// TIA Portal project "Elevator" (V16)

(* hardware
DEVICE "S71500/ET200MP station_1"  S7-1500 station
   slot 0: "Perfil soporte_0"  Rack  6ES7 590-1***0-0AA0
   slot 1: "PLC_1"  CPU 1511-1 PN  6ES7 511-1AK02-0AB0  V2.8
      slot 3: "Display de la CPU_1"  6ES7591-1AA00-0AA0
      slot 32768: "Interfaz PROFINET_1"  X1
         slot 32769: "Puerto_1"  X1 P1
         slot 32770: "Puerto_2"  X1 P2
      slot 34817: "Virtual CP interface port_1"  Virtual CP interface port  Virtual CP interface port
*)

// ===== PLC "PLC_1"  CPU 1511-1 PN =====

VAR_GLOBAL   // PLC tag table "Tabla de variables estándar"
   "Tag_1" AT %M0.0 : Bool;
   "Tag_2" AT %M0.1 : Bool;
   "Tag_3" AT %M200.0 : Bool;
END_VAR

DATA_BLOCK "Floor"   // DB1
{ S7_Optimized_Access := 'TRUE' }
VERSION : 0.1
   VAR
      Piso_1 : Real := 3166.0;
      Piso_2 : Real := 6332.0;
      Piso_3 : Real := 9498.0;
      Piso_4 : Real := 12664.0;
      Piso_5 : Real;
      Piso_6 : Real := -19000.0;
      PisoActual : Real := 3166.0;
      Floor_Command : Int := 0;
   END_VAR
BEGIN
END_DATA_BLOCK

ORGANIZATION_BLOCK "Main"   // OB1, LAD, ProgramCycle
TITLE = "Main Program Sweep (Cycle)"
{ S7_Optimized_Access := 'TRUE' }
VERSION : 0.1
   VAR_INPUT
      Initial_Call : Bool;   // Initial call of this OB
      Remanence : Bool;   // =True, if remanent data are available
   END_VAR
BEGIN

REGION Network 1
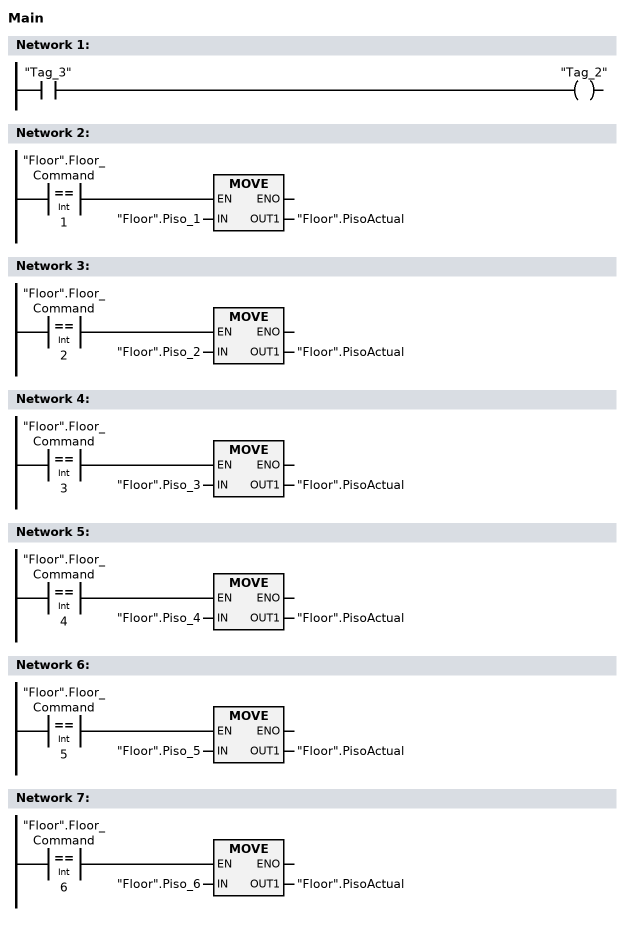
   RUNG wire#powerrail
      Contact( "Tag_3" )
      Coil( "Tag_2" )
   END_RUNG
   // the same network as SCL:
   "Tag_2" := "Tag_3";
END_REGION

REGION Network 2
   RUNG wire#powerrail
      { S7_Templates := "SrcType := Int" } EQ_Contact(in1 := "Floor".Floor_Command, in2 := 1)
      Move(in := "Floor".Piso_1, out1 => "Floor".PisoActual)
   END_RUNG
   // the same network as SCL:
   IF "Floor".Floor_Command = 1 THEN "Floor".PisoActual := "Floor".Piso_1; END_IF;
END_REGION

REGION Network 3
   RUNG wire#powerrail
      { S7_Templates := "SrcType := Int" } EQ_Contact(in1 := "Floor".Floor_Command, in2 := 2)
      Move(in := "Floor".Piso_2, out1 => "Floor".PisoActual)
   END_RUNG
   // the same network as SCL:
   IF "Floor".Floor_Command = 2 THEN "Floor".PisoActual := "Floor".Piso_2; END_IF;
END_REGION

REGION Network 4
   RUNG wire#powerrail
      { S7_Templates := "SrcType := Int" } EQ_Contact(in1 := "Floor".Floor_Command, in2 := 3)
      Move(in := "Floor".Piso_3, out1 => "Floor".PisoActual)
   END_RUNG
   // the same network as SCL:
   IF "Floor".Floor_Command = 3 THEN "Floor".PisoActual := "Floor".Piso_3; END_IF;
END_REGION

REGION Network 5
   RUNG wire#powerrail
      { S7_Templates := "SrcType := Int" } EQ_Contact(in1 := "Floor".Floor_Command, in2 := 4)
      Move(in := "Floor".Piso_4, out1 => "Floor".PisoActual)
   END_RUNG
   // the same network as SCL:
   IF "Floor".Floor_Command = 4 THEN "Floor".PisoActual := "Floor".Piso_4; END_IF;
END_REGION

REGION Network 6
   RUNG wire#powerrail
      { S7_Templates := "SrcType := Int" } EQ_Contact(in1 := "Floor".Floor_Command, in2 := 5)
      Move(in := "Floor".Piso_5, out1 => "Floor".PisoActual)
   END_RUNG
   // the same network as SCL:
   IF "Floor".Floor_Command = 5 THEN "Floor".PisoActual := "Floor".Piso_5; END_IF;
END_REGION

REGION Network 7
   RUNG wire#powerrail
      { S7_Templates := "SrcType := Int" } EQ_Contact(in1 := "Floor".Floor_Command, in2 := 6)
      Move(in := "Floor".Piso_6, out1 => "Floor".PisoActual)
   END_RUNG
   // the same network as SCL:
   IF "Floor".Floor_Command = 6 THEN "Floor".PisoActual := "Floor".Piso_6; END_IF;
END_REGION
END_ORGANIZATION_BLOCK